// TwinCAT 3 PLC project virtual_plc
// ProgramVersion: 3.1.4024.0
// libraries:
//   Tc2_Standard, * (Beckhoff Automation GmbH)
//   Tc2_System, * (Beckhoff Automation GmbH)
//   Tc3_Module, * (Beckhoff Automation GmbH)
// project tree:
//   / PlcTask.TcTTO
//   POUs/ Functieprogramma.TcPOU, GVL.TcGVL, TaskKoffieZetten.TcPOU, TaskWakkerWorden.TcPOU
// real-time tasks:
//   TASK PlcTask: cycle T#10ms, priority 20, ADS port 350
//   TASK Taak1: cycle T#20ms, priority 1, ADS port 351
//   TASK Taak2: cycle T#30ms, priority 21, ADS port 352

CONFIGURATION virtual_plc
    RESOURCE PLC ON TwinCAT3
        TASK PlcTask(INTERVAL := T#10ms, PRIORITY := 20);
        PROGRAM MAIN WITH PlcTask : MAIN;
    END_RESOURCE
END_CONFIGURATION

// ---- POUs/GVL.TcGVL

VAR_GLOBAL
    g_bWekTijd       : BOOL := FALSE;   // Wordt TRUE waneer het tijd is om wakker te worden
    g_bWakker         : BOOL := FALSE;   // Wordt TRUE als Task1 ziet dat je wakker bent
    g_bLampAan          : BOOL := FALSE;   // Wordt aangestuurd door TaskWakkerWorden
    g_bKoffieKlaar      : BOOL := FALSE;   // Wordt gebruikt in TaskKoffieZetten
    g_iSnoozeCounter    : INT := 0;        // Wordt aangepast en bijgehouden door TaskWakkerWorden
	g_WakkerWorden 	: BOOL;					// Houdt bij of de gebruiker al wakker moet worden
	g_KoffieZetten   : TON;					// Is de timer die bijhoud of de koffie klaar is
END_VAR

// ---- POUs/TaskWakkerWorden.TcPOU
VAR
    	
END_VAR


// Kijken of het tijd is om wakker te worden door de functie aan te roepen
GVL.g_WakkerWorden := TijdVanWakkerWorden(
                    ActueleUur := 7, 
                    ActueleMinuut := 0,
                    WekUur := 7,
                    WekMinuut := 0);

// Als het tijd is om wakker te worden GVL updaten
IF GVL.g_WakkerWorden THEN
    GVL.g_bWekTijd := TRUE;
    GVL.g_bLampAan := TRUE;

    // Wakker worden simuleren
    GVL.g_iSnoozeCounter := GVL.g_iSnoozeCounter + 1;

    IF GVL.g_iSnoozeCounter > 2 THEN
        GVL.g_bWakker := TRUE;
    END_IF
END_IF

// ---- POUs/TaskKoffieZetten.TcPOU
VAR
    
END_VAR


// Koffieapparaat aanzetten zodra gebruiker wakker is
IF GVL.g_bWakker THEN
    GVL.g_KoffieZetten(IN := TRUE, PT := T#10S);  // Koffie loopt voor 10 seconden
ELSE
    GVL.g_KoffieZetten(IN := FALSE);
END_IF

// Koffie is klaar zodra de timer klaar is
IF GVL.g_KoffieZetten.Q THEN
    GVL.g_bKoffieKlaar := TRUE;
END_IF

// ---- POUs/Functieprogramma.TcPOU
FUNCTION TijdVanWakkerWorden : BOOL
VAR_INPUT
    ActueleUur   : INT;
    ActueleMinuut : INT;
    WekUur      : INT;
    WekMinuut    : INT;
END_VAR



IF (ActueleUur = WekUur) AND (ActueleMinuut = Wekminuut) THEN
    TijdVanWakkerWorden := TRUE;
ELSE
    TijdVanWakkerWorden := FALSE;
END_IF

END_FUNCTION
